FUNCTION_BLOCK STR_Param
VAR_INPUT PERSISTENT
	val			: Strings.Str;
END_VAR

END_FUNCTION_BLOCK

(* stored: Version 1.1.0.1
   POU STR_Param: Id {5d3d2612-01dc-45ff-b31c-9b5719f131f7}, SpecialFunc None *)
